FUNCTION TryConvert_WORD_TO_TIME : BOOL
VAR_INPUT
	in : WORD;
	out : REFERENCE TO TIME;
END_VAR

out := WORD_TO_TIME(in);
TryConvert_WORD_TO_TIME := TRUE;

END_FUNCTION

(* stored: Version 1.1.0.1, ProductVersion 3.1.4024.12
   POU TryConvert_WORD_TO_TIME: Id {569e49e6-f48c-4aad-a432-339daf253e31}, SpecialFunc None *)
